# EPICS autosave request: iocBoot/ioc13idc/auto_settings.req
file "scaler_settings.req",             P=$(P), S=scaler1
file "Keithley2kDMM_mf10_settings.req", P=$(P), Dmm=DMM1
file "SR570preamp_settings.req",        P=$(P), A=A1
file "SR570preamp_settings.req",        P=$(P), A=A2
file "SR570preamp_settings.req",        P=$(P), A=A3
file "SR570preamp_settings.req",        P=$(P), A=A4
#file "SR570preamp_settings.req",        P=$(P), A=A5
#file "SR570preamp_settings.req",        P=$(P), A=A6
file "SR570preamp_settings.req",        P=$(P), A=B1
file "SR570preamp_settings.req",        P=$(P), A=B2
file "SR570preamp_settings.req",        P=$(P), A=B3
file "SR570preamp_settings.req",        P=$(P), A=B4
file "SIS38XX_settings.req",            P=$(P)SIS1:
file "Pelco_CM6700_settings.req",       P=$(P), R=Pelco1
##file "icb_adc_settings.req",            P=$(P), ADC=adc1
#file "icb_amp_settings.req",            P=$(P), AMP=amp1
#file "icb_hvps_settings.req",           P=$(P), HVPS=hvps1
##file "mca_settings.req",                P=$(P), M=aim_adc1
##file "mca_settings.req",                P=$(P), M=aim_mcs1
file "mca_settings.req",                P=$(P), M=mip330_1
file "mca_settings.req",                P=$(P), M=mip330_2
file "mca_settings.req",                P=$(P), M=mip330_3
file "mca_settings.req",                P=$(P), M=mip330_4
file "mca_settings.req",                P=$(P), M=mip330_5
file "mca_settings.req",                P=$(P), M=mip330_6
file "scan_settings.req",               P=$(P), S=scan1
file "scan_settings.req",               P=$(P), S=scan2
file "scan_settings.req",               P=$(P), S=scan3
file "scan_settings.req",               P=$(P), S=scan4
file "saveData_settings.req",           P=$(P)
file "sca_window.req",                  P=$(P), SCA=BEDE
file "filterDrive.req",                 P=$(P), R=filter:
file "filterBladeNoSensor.req",         P=$(P), R=filter:, N=1
file "filterBladeNoSensor.req",         P=$(P), R=filter:, N=2
file "filterBladeNoSensor.req",         P=$(P), R=filter:, N=3
file "filterBladeNoSensor.req",         P=$(P), R=filter:, N=4
file "filterBladeNoSensor.req",         P=$(P), R=filter:, N=5
file "filterBladeNoSensor.req",         P=$(P), R=filter:, N=6
file "filterBladeNoSensor.req",         P=$(P), R=filter:, N=7
file "filterBladeNoSensor.req",         P=$(P), R=filter:, N=8
file "userArrayCalcs10_settings.req",   P=$(P)
file "userStringCalcs10_settings.req",  P=$(P)
file "userTransforms10_settings.req",   P=$(P)
file "CARS_24_motor_settings.req",      P=$(P)
file "CARS_motor_settings.req",         P=$(P), M=m41
file "CARS_motor_settings.req",         P=$(P), M=m42
file "CARS_motor_settings.req",         P=$(P), M=m43
file "CARS_motor_settings.req",         P=$(P), M=m44
file "CARS_motor_settings.req",         P=$(P), M=m45
file "CARS_motor_settings.req",         P=$(P), M=m46
file "CARS_motor_settings.req",         P=$(P), M=m47
file "CARS_motor_settings.req",         P=$(P), M=m48
file "CARS_motor_settings.req",         P=$(P), M=m49
file "CARS_motor_settings.req",         P=$(P), M=m50
file "CARS_motor_settings.req",         P=$(P), M=m51
file "CARS_motor_settings.req",         P=$(P), M=m52
file "CARS_motor_settings.req",         P=$(P), M=m53
file "CARS_motor_settings.req",         P=$(P), M=m54
file "CARS_motor_settings.req",         P=$(P), M=m55
file "CARS_motor_settings.req",         P=$(P), M=m56
file "CARS_motor_settings.req",         P=$(P), M=m57
file "CARS_motor_settings.req",         P=$(P), M=m58
file "CARS_motor_settings.req",         P=$(P), M=m59
file "CARS_motor_settings.req",         P=$(P), M=m60
file "CARS_motor_settings.req",         P=$(P), M=m61
file "CARS_motor_settings.req",         P=$(P), M=m62
file "CARS_motor_settings.req",         P=$(P), M=m63
file "CARS_motor_settings.req",         P=$(P), M=m64
